# EPICS autosave request: iocBoot/ioc13GasLoading/auto_positions.req
file "CARS_motor_positions.req",         P=$(P), M=m3
file "CARS_motor_positions.req",         P=$(P), M=m4
file "CARS_motor_positions.req",         P=$(P), M=m5
file "CARS_motor_positions.req",         P=$(P), M=m7
file "CARS_motor_positions.req",         P=$(P), M=m8
